// Block: DecoilersHRot_PERS

DATA_BLOCK DecoilersHRot_PERS
VERSION : 0.1
   NON_RETAIN
   VAR
      PersistentValues : Struct
         Par : Struct
            TraslationAx : Positioning_DOL_Machine_Par;
            TraslationEnc : PosFbk_RTN;
            Traslation_AutSpeed : Real;
         END_STRUCT;
         Ax_Pers : Positioning_DOL_Machine_Pers_Data;
      END_STRUCT;
   END_VAR

BEGIN
   // No initialization required
END_DATA_BLOCK
